{attribute 'qualified_only'}
{attribute 'strict'}
TYPE E_DIRECTION :
(
	NEGATIVE := 1,
	POSITIVE
);
END_TYPE

(* stored: Version 1.1.0.1, ProductVersion 3.1.4022.16
   DUT E_DIRECTION: Id {40fffe57-8c26-4457-870a-0963b43b7bac} *)
